{attribute 'monitoring' := 'call'}
PROPERTY Simulated : BOOL
GET
END_GET
END_PROPERTY

{attribute 'monitoring' := 'call'}
PROPERTY Vdc24Okay : BOOL
GET
END_GET
END_PROPERTY

{attribute 'monitoring' := 'call'}
PROPERTY Vdc48Okay : BOOL
GET
END_GET
END_PROPERTY

END_FUNCTION_BLOCK

// _Internal/NullObjects/NullXtsSystemTasks
{attribute 'no_explicit_call' := 'This FB is a CLASS and must be accessed using methods or properties'}
{attribute 'conditionalshow'}
{warning disable C0094}
FUNCTION_BLOCK NullXtsSystemTasks IMPLEMENTS I_XtsTaskCollection, I_NullObject
VAR
END_VAR

METHOD AddTask : BOOL
VAR_INPUT
	Task	: I_XtsTask;
END_VAR
END_METHOD

METHOD CyclicLogic
END_METHOD

METHOD GetTaskById : I_XtsTask
VAR_INPUT
	TaskId	: XtsSystemTaskId;
END_VAR
GetTaskById := NullObjects.XtsTask;
END_METHOD

METHOD GetTaskByName : I_XtsTask
VAR_INPUT
	Name	: T_MaxString;
END_VAR
GetTaskByName := NullObjects.XtsTask;
END_METHOD

METHOD RemoveTaskById
VAR_INPUT
	TaskId	: XtsSystemTaskId;
END_VAR
END_METHOD

METHOD RemoveTaskByInstance
VAR_INPUT
	Task	: I_XtsTask;
END_VAR
END_METHOD

END_FUNCTION_BLOCK

// _Internal/NullObjects/NullXtsTrackCollection
{attribute 'no_explicit_call' := 'This FB is a CLASS and must be accessed using methods or properties'}
{attribute 'conditionalshow'}
{warning disable C0094}
{warning disable C0568}
FUNCTION_BLOCK NullXtsTrackCollection IMPLEMENTS I_XtsTrackCollection, I_NullObject
VAR
END_VAR

METHOD Clear
END_METHOD

PROPERTY Count : UDINT
GET
END_GET
END_PROPERTY

{attribute 'hide'}
METHOD Create : BOOL
VAR_INPUT
	NumberOfTracks : UINT;
END_VAR
END_METHOD

{attribute 'monitoring' := 'call'}
PROPERTY Current : I_XtsTrack
GET
Current := NullObjects.XtsTrack;
END_GET
END_PROPERTY

{attribute 'monitoring' := 'call'}
PROPERTY CurrentIndex : UDINT
GET
END_GET
END_PROPERTY

METHOD GetById : I_XtsTrack
VAR_INPUT
	TrackId : UDINT;
END_VAR
GetById := NullObjects.XtsTrack;
END_METHOD

METHOD GetByOtcid : I_XtsTrack
VAR_INPUT
	TrackOtcid : OTCID;
END_VAR
GetByOtcid := NullObjects.XtsTrack;
END_METHOD

{attribute 'monitoring' := 'call'}
PROPERTY IsEmpty : BOOL
GET
END_GET
END_PROPERTY

PROPERTY MoveToNext : BOOL
GET
END_GET
END_PROPERTY

METHOD ResetIterator
END_METHOD

END_FUNCTION_BLOCK

// _Internal/NullObjects/NullXtsZone
{attribute 'no_explicit_call' := 'This FB is a CLASS and must be accessed using methods or properties'}
{attribute 'conditionalshow'}
{warning disable C0094}
{warning disable C0568}
FUNCTION_BLOCK NullXtsZone IMPLEMENTS I_XtsZone, I_NullObject
VAR
END_VAR

METHOD Accept
VAR_INPUT
	ComponentVisitor	: Core.I_ComponentVisitor;
END_VAR
END_METHOD

METHOD AcceptMoverVisitor
VAR_INPUT
	MoverVisitor : I_XtsMoverVisitor;
END_VAR
END_METHOD

METHOD AcceptXtsZoneVisitor
VAR_INPUT
	ZoneVisitor : I_XtsZoneVisitor;
END_VAR
END_METHOD

{attribute 'monitoring':='call'}
PROPERTY CommandLog : I_XtsLocalLog
GET
CommandLog := NullObjects.MechatronicsLocalLog;
END_GET
END_PROPERTY

METHOD DeregisterWithParent
VAR_INPUT
	Parent	: Core.I_ContainComponents;
END_VAR
END_METHOD

PROPERTY EndPosition : LREAL
GET
END_GET
SET
END_SET
END_PROPERTY

//Select the Nth Mover in the Zone
METHOD GetSortedMover : I_XtsMover
VAR_INPUT
	Index	  : UDINT; // 1 based index
	Direction : Tc3_Mc3Definitions.MC_DIRECTION := Tc3_Mc3Definitions.MC_DIRECTION.mcDirectionPositive; //Direction to fetch from
END_VAR
END_METHOD

METHOD IsMoverInZone : BOOL
VAR_INPUT
	Mover : I_XtsMover;
END_VAR
END_METHOD

PROPERTY Length : LREAL
GET
END_GET
END_PROPERTY

PROPERTY MonitoredMovers : I_XtsMoverCollection
SET
END_SET
END_PROPERTY

PROPERTY Movers : I_XtsMoverEnumerator
GET
Movers := NullObjects.XtsMoverList;
END_GET
END_PROPERTY

PROPERTY Name : Core.T_MaxString
GET
Name := 'Null Xts Zone';
END_GET
SET
END_SET
END_PROPERTY

METHOD RegisterWithParent
VAR_INPUT
	Parent	: Core.I_ContainComponents;
END_VAR
END_METHOD

PROPERTY StartPosition : LREAL
GET
END_GET
SET
END_SET
END_PROPERTY

{attribute 'monitoring':='call'}
PROPERTY Status : I_XtsZoneStatus
GET
Status := NullObjects.XtsZoneStatus;
END_GET
END_PROPERTY

PROPERTY TracePublisher : I_XtsTracePublisher
GET
TracePublisher := NullObjects.MechatronicsTracePublisher;
END_GET
END_PROPERTY

END_FUNCTION_BLOCK

// _Internal/Zone/Status/XtsZoneStatus
{attribute 'no_explicit_call' := 'This FB is a CLASS and must be accessed using methods or properties'}
FUNCTION_BLOCK XtsZoneStatus IMPLEMENTS I_XtsZoneStatus
VAR
	_Zone	: I_XtsZone;
	_Movers : I_XtsMoverCollection;
END_VAR

//FB_Init is always available implicitly and it is used primarily for initialization.

//The return value is not evaluated. For a specific influence, you can also declare the

//methods explicitly and provide additional code there with the standard initialization

//code. You can evaluate the return value.
METHOD FB_Init : BOOL
VAR_INPUT
	bInitRetains : BOOL; // TRUE: the retain variables are initialized (reset warm / reset cold)
	bInCopyCode	 : BOOL; // TRUE: the instance will be copied to the copy code afterward (online change)   
	Zone		 : I_XtsZone;
END_VAR
_Zone := Zone;
END_METHOD

{attribute 'monitoring' := 'call'}
//Number of Movers Currently in Zone
PROPERTY NumberOfMoversInZone : UDINT
GET
NumberOfMoversInZone := _Movers.Count;
END_GET
END_PROPERTY

METHOD SetMoverCollection
VAR_INPUT
	MoverCollection : I_XtsMoverCollection;
END_VAR
_Movers := MoverCollection;
END_METHOD

END_FUNCTION_BLOCK

// _Internal/NullObjects/NullXtsZoneStatus
{attribute 'no_explicit_call' := 'This FB is a CLASS and must be accessed using methods or properties'}
{attribute 'conditionalshow'}
{warning disable C0094}
FUNCTION_BLOCK NullXtsZoneStatus IMPLEMENTS I_XtsZoneStatus, I_NullObject
VAR
END_VAR

{attribute 'monitoring' := 'call'}
PROPERTY NumberOfMoversInZone : UDINT
GET
END_GET
END_PROPERTY

END_FUNCTION_BLOCK

// _Internal/NullObjects/NullZoneCollection
{attribute 'no_explicit_call' := 'This FB is a CLASS and must be accessed using methods or properties'}
{attribute 'conditionalshow'}
{warning disable C0094}
{warning disable C0568}
FUNCTION_BLOCK NullZoneCollection IMPLEMENTS I_XtsZoneCollection, I_NullObject
VAR
END_VAR

METHOD AddItem
VAR_INPUT
	Zone	: I_XtsZone;
END_VAR
END_METHOD

METHOD Clear
END_METHOD

PROPERTY Count : UDINT
GET
END_GET
END_PROPERTY

PROPERTY Current : I_XtsZone
GET
Current := NullObjects.XtsZone;
END_GET
END_PROPERTY

PROPERTY CurrentItem : UDINT
GET
END_GET
END_PROPERTY

{attribute 'monitoring' := 'call'}
PROPERTY IsEmpty : BOOL
GET
END_GET
END_PROPERTY

PROPERTY MoveToNext : BOOL
GET
END_GET
END_PROPERTY

METHOD Remove
VAR_INPUT
	Zone	: I_XtsZone;
END_VAR
END_METHOD

METHOD ResetIterator
END_METHOD

END_FUNCTION_BLOCK

// XtsZone/XtsZone
{attribute 'no_explicit_call' := 'This FB is a CLASS and must be accessed using methods or properties'}
FUNCTION_BLOCK XtsZone EXTENDS CyclicComponent IMPLEMENTS I_XtsZone
VAR
	{attribute 'hide'}
	_Status		: XtsZoneStatus(THIS^);
	_Properties : _DefaultZonePropertyBackers;
	{attribute 'hide'}
	_LocalLogger : XtsLocalLogger;
	{attribute 'hide'}
	_Logger				: XtsTracePublisher;
	_DimensionChecker	: SingleDimensionChecker(_Properties.SingleDimensionBacker);
	_MoverComparer		: MoverZoneDistanceComparer(_Properties.SingleDimensionBacker);
	_DefaultZoneMonitor : ZoneMonitor(_DimensionChecker, _MoverComparer, _Properties.SingleDimensionBacker, _Logger);
	_ZoneMonitor		: I_ZoneMonitor := _DefaultZoneMonitor;
	{attribute 'hide'}
	LogSource : TraceSourceInfo;
	{attribute 'hide'}
	LogMessage : TraceMessageInfo;
END_VAR

//FB_Init is always available implicitly and it is used primarily for initialization.

//The return value is not evaluated. For a specific influence, you can also declare the

//methods explicitly and provide additional code there with the standard initialization

//code. You can evaluate the return value.
METHOD FB_Init : BOOL
VAR_INPUT
	bInitRetains	: BOOL;				 // TRUE: the retain variables are initialized (reset warm / reset cold)
	bInCopyCode		: BOOL;				 // TRUE: the instance will be copied to the copy code afterward (online change)   
	Name			: T_MaxString;		 //Name of the Zone
	MonitoredMovers : I_XtsMoverCollection; //Collection of Movers for the Zone to monitor
	StartPosition	: LREAL := 0;		 //Start position of the Zone in mm
	EndPosition		: LREAL := 0;		 //End position of the Zone in mm
	System			: I_ContainXtsZones; //XtsSystem to self register to
END_VAR
_ZoneMonitor.MonitoredMovers := MonitoredMovers;
LogSource.SourceName		 := 'Zone Object';
_Logger.Subscribe(_LocalLogger);
IF XtsCoreParameters.TcEventLoggerEnabled THEN
	_Logger.Subscribe(XtsTrace.EventLogger);
END_IF

_Status.SetMoverCollection(_ZoneMonitor.Movers);
THIS^.StartPosition := StartPosition;
THIS^.EndPosition	:= EndPosition;
IF System <> 0 THEN
	System.Zones.AddItem(THIS^);
	RegisterWithParent(System);
END_IF
END_METHOD

{attribute 'monitoring':='call'}
//End Position of the Zone in mm
PROPERTY EndPosition : LREAL
GET
EndPosition := _Properties.SingleDimensionBacker.EndPosition;
END_GET
SET
_Properties.SingleDimensionBacker.EndPosition := EndPosition;
END_SET
END_PROPERTY

{attribute 'monitoring':='call'}
//Start Position of the Zone in mm
PROPERTY StartPosition : LREAL
GET
StartPosition := _Properties.SingleDimensionBacker.StartPosition;
END_GET
SET
_Properties.SingleDimensionBacker.StartPosition := StartPosition;
END_SET
END_PROPERTY

{attribute 'monitoring':='call'}
PROPERTY CommandLog : I_XtsLocalLog
GET
CommandLog := _LocalLogger;
END_GET
END_PROPERTY

PROPERTY TracePublisher : I_XtsTracePublisher
GET
TracePublisher := _Logger;
END_GET
END_PROPERTY

METHOD AcceptMoverVisitor
VAR_INPUT
	MoverVisitor	: I_XtsMoverVisitor;
END_VAR
_ZoneMonitor.Movers.AcceptMoverVisitor(MoverVisitor);
END_METHOD

METHOD AcceptXtsZoneVisitor
VAR_INPUT
	ZoneVisitor : I_XtsZoneVisitor;
END_VAR
ZoneVisitor.VisitZone(THIS^);
END_METHOD

METHOD CyclicLogic
VAR
	Mover : I_XtsMover;
END_VAR
_ZoneMonitor.CyclicLogic();
END_METHOD

//Select the Nth Mover in the Zone
METHOD GetSortedMover : I_XtsMover
VAR_INPUT
	Index	  : UDINT; // 1 based index
	Direction : Tc3_Mc3Definitions.MC_DIRECTION := Tc3_Mc3Definitions.MC_DIRECTION.mcDirectionPositive; //Direction to fetch from
END_VAR
VAR
	DesiredIndex : UDINT;
END_VAR
GetSortedMover := NullObjects.XtsMover;
IF Index <= 0 OR Index > _ZoneMonitor.Movers.Count THEN
	LogMessage.Message	 := 'GetSortedMover Requested Index Out of bounds';
	LogMessage.Severity	 := 2;
	LogMessage.MessageId := E_XtsLogMessage.ZoneMoverErrorGetSortedIndexOOB;
	_Logger.LogMessageInstance(LogSource, LogMessage);
	RETURN;
END_IF

IF Direction = Tc3_Mc3Definitions.MC_Direction.mcDirectionNegative THEN
	DesiredIndex := _ZoneMonitor.Movers.Count - Index;
ELSE
	DesiredIndex := Index - 1;
END_IF

GetSortedMover := _ZoneMonitor.Movers.GetAtIndex(DesiredIndex);
END_METHOD

//Check if Mover is currently in Zone
METHOD IsMoverInZone : BOOL
VAR_INPUT
	Mover : I_XtsMover; //Mover to check
END_VAR
IsMoverInZone := _ZoneMonitor.Movers.Contains(Mover);
END_METHOD

//Movers currently monitored by Zone
PROPERTY MonitoredMovers : I_XtsMoverCollection
SET
_ZoneMonitor.MonitoredMovers := MonitoredMovers;
END_SET
END_PROPERTY

//Movers currently in the Zone
PROPERTY Movers : I_XtsMoverEnumerator
GET
Movers := _ZoneMonitor.Movers;
END_GET
END_PROPERTY

{attribute 'monitoring':='call'}
PROPERTY Status : I_XtsZoneStatus
GET
Status := _Status;
END_GET
END_PROPERTY

END_FUNCTION_BLOCK

// _Internal/Zone/Properties/_DefaultZonePropertyBackers
{attribute 'no_explicit_call' := 'This FB is a CLASS and must be accessed using methods or properties'}
FUNCTION_BLOCK _DefaultZonePropertyBackers
VAR
	_DefaultSingleDimensionZone : SingleDimensionZone;
	//
	_SingleDimensionZone : I_SingleDimensionZone := _DefaultSingleDimensionZone;
END_VAR

{attribute 'monitoring':='call'}
PROPERTY SingleDimensionBacker : I_SingleDimensionZone
GET
SingleDimensionBacker := _SingleDimensionZone;
END_GET
SET
_SingleDimensionZone := SingleDimensionBacker;
END_SET
END_PROPERTY

END_FUNCTION_BLOCK

// _Internal/Zone/Properties/SingleDimensionZone
{attribute 'no_explicit_call' := 'This FB is a CLASS and must be accessed using methods or properties'}
FUNCTION_BLOCK SingleDimensionZone IMPLEMENTS I_SingleDimensionZone
VAR
	_StartPosition : LREAL;
	_EndPosition   : LREAL;
END_VAR

{attribute 'monitoring':='call'}
PROPERTY EndPosition : LREAL
GET
EndPosition := _EndPosition;
END_GET
SET
_EndPosition := EndPosition;
END_SET
END_PROPERTY

{attribute 'monitoring':='call'}
PROPERTY StartPosition : LREAL
GET
StartPosition := _StartPosition;
END_GET
SET
_StartPosition := StartPosition;
END_SET
END_PROPERTY

END_FUNCTION_BLOCK

// _Internal/Zone/SingleDimensionChecker
{attribute 'no_explicit_call' := 'This FB is a CLASS and must be accessed using methods or properties'}
{attribute 'conditional_show'}
FUNCTION_BLOCK SingleDimensionChecker IMPLEMENTS I_MoverInPositionChecker
VAR
	_Dimensions : I_SingleDimensionZone;
END_VAR

//FB_Init is always available implicitly and it is used primarily for initialization.

//The return value is not evaluated. For a specific influence, you can also declare the

//methods explicitly and provide additional code there with the standard initialization

//code. You can evaluate the return value.
METHOD FB_Init : BOOL
VAR_INPUT
	bInitRetains : BOOL; // TRUE: the retain variables are initialized (reset warm / reset cold)
	bInCopyCode	 : BOOL; // TRUE: the instance will be copied to the copy code afterward (online change)  
	Dimensions	 : I_SingleDimensionZone;
END_VAR
_Dimensions := Dimensions;
END_METHOD

METHOD IsMoverInPosition : BOOL
VAR_INPUT
	Mover : I_XtsMover;
END_VAR

VAR
	startPosition : LREAL;
	endPosition	  : LREAL;
	tmp : LREAL;
END_VAR
startPosition := _Dimensions.StartPosition;
endPosition	  := _Dimensions.EndPosition;
IF Mover.Status.CurrentTrack.Length <> 0 THEN
	startPosition := startPosition - Mover.Status.CurrentTrack.Length * TRUNC(_Dimensions.StartPosition / Mover.Status.CurrentTrack.Length);
	IF startPosition < 0.0 THEN
		startPosition := startPosition + Mover.Status.CurrentTrack.Length;
	END_IF

	endPosition := endPosition - Mover.Status.CurrentTrack.Length * TRUNC(_Dimensions.EndPosition / Mover.Status.CurrentTrack.Length);
	IF endPosition < 0.0 THEN
		endPosition := endPosition + Mover.Status.CurrentTrack.Length;
	END_IF
END_IF

IF startPosition < endPosition THEN
	IsMoverInPosition := Mover.Position > startPosition AND Mover.Position < endPosition;
ELSE
	IsMoverInPosition := Mover.Position > startPosition OR Mover.Position < endPosition;
END_IF
END_METHOD

END_FUNCTION_BLOCK

// _Internal/Zone/Interfaces/I_MoverInPositionChecker
INTERFACE I_MoverInPositionChecker EXTENDS I_Base

METHOD IsMoverInPosition : BOOL
VAR_INPUT
	Mover : I_XtsMover;
END_VAR
END_METHOD

END_INTERFACE

// _Internal/Zone/MoverZoneDistanceComparer
{attribute 'no_explicit_call' := 'This FB is a CLASS and must be accessed using methods or properties'}
{attribute 'conditional_show'}
FUNCTION_BLOCK MoverZoneDistanceComparer IMPLEMENTS I_XtsMoverComparer
VAR
	_ZoneDimensions : I_SingleDimensionZone;
END_VAR

METHOD Compare : SINT
VAR_INPUT
	Mover1 : I_XtsMover;
	Mover2 : I_XtsMover;
END_VAR

VAR
	Mover1Distance : LREAL;
	Mover2Distance : LREAL;
END_VAR
Mover1Distance := MoverDistance(_ZoneDimensions.StartPosition, Mover1.Position, Mover1.Status.CurrentTrack.Length);
Mover2Distance := MoverDistance(_ZoneDimensions.StartPosition, Mover2.Position, Mover2.Status.CurrentTrack.Length);
IF Mover1Distance < Mover2Distance THEN
	Compare := -1;
ELSIF Mover1Distance > Mover2Distance THEN
	Compare := 1;
ELSE
	Compare := 0;
END_IF
END_METHOD

//FB_Init is always available implicitly and it is used primarily for initialization.
//The return value is not evaluated. For a specific influence, you can also declare the
//methods explicitly and provide additional code there with the standard initialization
//code. You can evaluate the return value.
METHOD FB_Init: BOOL
VAR_INPUT
    bInitRetains: BOOL; // TRUE: the retain variables are initialized (reset warm / reset cold)
    bInCopyCode: BOOL;  // TRUE: the instance will be copied to the copy code afterward (online change)   
	Dimensions : I_SingleDimensionZone;
END_VAR
_ZoneDimensions := Dimensions;
END_METHOD

END_FUNCTION_BLOCK

// _Internal/Zone/Interfaces/I_XtsMoverComparer
INTERFACE I_XtsMoverComparer EXTENDS I_Base

METHOD Compare : SINT
VAR_INPUT
	Mover1 : I_XtsMover;
	Mover2 : I_XtsMover;
END_VAR
END_METHOD

END_INTERFACE

// _Internal/Zone/MoverDistance
FUNCTION MoverDistance : LREAL
VAR_INPUT
	StartPosition : LREAL;
	MoverPosition : LREAL;
	TrackLength	  : LREAL;
END_VAR

VAR
	NormalizedStart : LREAL;
	Distance		: LREAL;
END_VAR

IF TrackLength = 0 THEN
	MoverDistance := 0;
	RETURN;
END_IF

NormalizedStart := StartPosition - TrackLength * TRUNC(StartPosition / TrackLength);
IF normalizedStart < 0 THEN
	NormalizedStart := NormalizedStart + TrackLength;
END_IF;

Distance := MoverPosition - NormalizedStart;
IF Distance < 0 THEN
	Distance := Distance + TrackLength;
END_IF;

MoverDistance := Distance;

END_FUNCTION

// _Internal/Zone/ZoneMonitor
{attribute 'no_explicit_call' := 'This FB is a CLASS and must be accessed using methods or properties'}
{attribute 'conditional_show'}
FUNCTION_BLOCK ZoneMonitor IMPLEMENTS I_ZoneMonitor
VAR
	_DefaultCurrentMovers : XtsMoverList;
	_CurrentMovers		  : I_XtsMoverList := _DefaultCurrentMovers;
	_MoverChecker		  : I_MoverInPositionChecker;
	_MonitoredMovers	  : I_XtsMoverCollection;
	_ZoneComparer		  : I_XtsMoverComparer;
	_ZoneDimensions		  : I_SingleDimensionZone;
	_Logger				  : I_XtsLogger;
	LogSource			  : TraceSourceInfo;
	LogMessage			  : TraceMessageInfo;
END_VAR

METHOD CyclicLogic
VAR
	Mover				   : I_XtsMover;
	inPosition			   : BOOL;
	inCollection		   : BOOL;
	additionIndex		   : UDINT;
	CompareResults		   : SINT;
	EntranceEvent		   : E_ThresholdEvent;
	ExitEvent			   : E_ThresholdEvent;
	ThresholdEventOccurred : BOOL;
END_VAR
_MonitoredMovers.ResetIterator();
WHILE _MonitoredMovers.MoveToNext DO
	__QUERYINTERFACE(_MonitoredMovers.Current, Mover);
	IF Mover.Status.CurrentTrack.Length = 0 THEN
		LogMessage.MessageId := E_XtsLogMessage.ZoneMoverErrorTrackLengthZero;
		LogMessage.Message	 := CONCAT(Mover.Name, ' current Track Length 0 unable to add to track');
		LogMessage.Severity	 := 3;
		_Logger.LogMessageInstance(LogSource, LogMessage);
		CONTINUE;
	END_IF

	inPosition := _MoverChecker.IsMoverInPosition(Mover);

	//Need to check if crossed the threshold of the exit or the entrance
	EntranceEvent		   := CheckForThresholdEvent(Mover, _ZoneDimensions.StartPosition);
	ExitEvent			   := CheckForThresholdEvent(Mover, _ZoneDimensions.EndPosition);
	ThresholdEventOccurred := (EntranceEvent <> E_ThresholdEvent.NoEvent) AND (ExitEvent <> E_ThresholdEvent.NoEvent);
	inCollection		   := _CurrentMovers.Contains(Mover);
	IF NOT inPosition AND inCollection THEN
		_CurrentMovers.Remove(Mover);
		CONTINUE;
	END_IF

	//Adds the Mover into the collection sorted by Position Descending
	IF inPosition AND NOT inCollection THEN
		_CurrentMovers.ResetIterator();
		WHILE _CurrentMovers.MoveToNext DO
			CompareResults := _ZoneComparer.Compare(Mover, _CurrentMovers.Current);
			IF CompareResults < 0 THEN //Mover 1 is closer to Start
				additionIndex := _CurrentMovers.CurrentItem - 1;
				EXIT;
			ELSIF CompareResults > 0 THEN //Mover 2 is closer to Start
				additionIndex := _CurrentMovers.CurrentItem;
			ELSE //Movers are equadistant, should never happen. Only realistically happens if TrackLength = 0

				//
			END_IF
		END_WHILE

		_CurrentMovers.InsertAtIndex(Mover, additionIndex);
	ELSIF ThresholdEventOccurred AND inCollection THEN
		(*Search the Collection to find the new index
			Remove from old index
			Add to new*)
		_CurrentMovers.ResetIterator();
		WHILE _CurrentMovers.MoveToNext DO
			CompareResults := _ZoneComparer.Compare(Mover, _CurrentMovers.Current);
			IF CompareResults < 0 THEN //Mover 1 is closer to Start
				additionIndex := _CurrentMovers.CurrentItem - 1;
				EXIT;
			ELSIF CompareResults > 0 THEN //Mover 2 is closer to Start
				additionIndex := _CurrentMovers.CurrentItem;
			ELSE //Movers are equadistant, should never happen. Only realistically happens if TrackLength = 0

				//
			END_IF
		END_WHILE

		_CurrentMovers.Remove(Mover);
		_CurrentMovers.InsertAtIndex(Mover, additionIndex);
	END_IF
END_WHILE
END_METHOD

//FB_Init is always available implicitly and it is used primarily for initialization.

//The return value is not evaluated. For a specific influence, you can also declare the

//methods explicitly and provide additional code there with the standard initialization

//code. You can evaluate the return value.
METHOD FB_Init : BOOL
VAR_INPUT
	bInitRetains	: BOOL; // TRUE: the retain variables are initialized (reset warm / reset cold)
	bInCopyCode		: BOOL; // TRUE: the instance will be copied to the copy code afterward (online change)   
	PositionChecker : I_MoverInPositionChecker;
	ZoneComparer	: I_XtsMoverComparer;
	ZoneDimensions	: I_SingleDimensionZone;
	Logger			: I_XtsLogger;
END_VAR
_MoverChecker		 := PositionChecker;
_ZoneComparer		 := ZoneComparer;
_Logger				 := Logger;
_ZoneDimensions		 := ZoneDimensions;
LogSource.SourceName := 'ZoneMonitor';
END_METHOD

PROPERTY MonitoredMovers : I_XtsMoverCollection
SET
_MonitoredMovers := MonitoredMovers;
END_SET
END_PROPERTY

{attribute 'monitoring':='call'}
PROPERTY Movers : I_XtsMoverList
GET
Movers := _CurrentMovers;
END_GET
END_PROPERTY

END_FUNCTION_BLOCK

// _Internal/Zone/Interfaces/I_ZoneMonitor
INTERFACE I_ZoneMonitor EXTENDS I_Base, I_Cyclic, I_MonitorsMovers, I_ContainXtsMoverList

END_INTERFACE

// _Internal/Peeker/Interfaces/I_XtsModuleCollectionPeeker
INTERFACE I_XtsModuleCollectionPeeker EXTENDS I_Base

METHOD SetCollection
VAR_INPUT
	NewCollection  : I_XtsModuleCollection;
	CollectionName : T_MaxString := 'A Collection';
END_VAR
END_METHOD

END_INTERFACE

// _Internal/Peeker/Interfaces/I_XtsMoverCollectionPeeker
INTERFACE I_XtsMoverCollectionPeeker EXTENDS I_Base

METHOD SetCollection
VAR_INPUT
	NewCollection  : I_XtsMoverCollection;
	CollectionName : T_MaxString := 'A Collection';
END_VAR
END_METHOD

END_INTERFACE

// _Internal/Peeker/Interfaces/I_XtsPartCollectionPeeker
INTERFACE I_XtsPartCollectionPeeker EXTENDS I_Base

METHOD SetCollection
VAR_INPUT
	NewCollection  : I_XtsPartCollection;
	CollectionName : T_MaxString := 'A Collection';
END_VAR
END_METHOD

END_INTERFACE

// _Internal/Peeker/Interfaces/I_XtsPositionTriggerCollectionPeeker
INTERFACE I_XtsPositionTriggerCollectionPeeker EXTENDS I_Base

METHOD SetCollection
VAR_INPUT
	NewCollection  : I_XtsPositionTriggerCollection;
	CollectionName : T_MaxString := 'A Collection';
END_VAR
END_METHOD

END_INTERFACE

// _Internal/Peeker/Interfaces/I_XtsStationCollectionPeeker
INTERFACE I_XtsStationCollectionPeeker EXTENDS I_Base

METHOD SetCollection
VAR_INPUT
	NewCollection  : I_XtsStationCollection;
	CollectionName : T_MaxString := 'A Collection';
END_VAR
END_METHOD

END_INTERFACE

// _Internal/Peeker/Interfaces/I_XtsZoneCollectionPeeker
INTERFACE I_XtsZoneCollectionPeeker EXTENDS I_Base

METHOD SetCollection
VAR_INPUT
	NewCollection  : I_XtsZoneCollection;
	CollectionName : T_MaxString := 'A Collection';
END_VAR
END_METHOD

END_INTERFACE

// _Internal/Station/Interfaces/I_StationTaskCollection
INTERFACE I_StationTaskCollection EXTENDS I_Base

END_INTERFACE

// _Internal/Station/MoverMonitorTask
{attribute 'no_explicit_call' := 'This FB is a CLASS and must be accessed using methods or properties'}
FUNCTION_BLOCK MoverMonitorTask IMPLEMENTS I_MoverMonitor
VAR
	_MonitoredMovers  : I_XtsMoverCollection;
	_CurrentMover	  : I_XtsMover := NullObjects.XtsMover;
	_RemoveCollection : XtsMoverCollection;
	_Station		  : I_XtsStation;
	{attribute 'hide'}
	_Logger : I_XtsLogger;
	{attribute 'hide'}
	LogSource : TraceSourceInfo;
	{attribute 'hide'}
	LogMessage : TraceMessageInfo;
END_VAR

METHOD CyclicLogic
VAR
	Mover	  : I_XtsMover;
	NullMover : I_XtsMover;
END_VAR
_MonitoredMovers.ResetIterator();
WHILE _MonitoredMovers.MoveToNext DO
	Mover := _MonitoredMovers.Current;
	IF Mover.CurrentTask.TaskId <> MoverTaskID.MOVE_TO_STATION OR Mover.Status.CommandedStation <> _Station THEN
		_RemoveCollection.AddItem(Mover);
		CONTINUE;
	END_IF

	NullMover := NullObjects.XtsMover;
	IF Mover.InPosition AND _CurrentMover = NullMover THEN
		_CurrentMover		 := Mover;
		LogMessage.Message	 := CONCAT(Mover.Name, ' arrived at station');
		LogMessage.MessageId := E_XtsLogMessage.StationMoverArrived;
		LogMessage.Severity	 := 0;
		_Logger.LogMessageInstance(LogSource, LogMessage);
		EXIT;
	END_IF
END_WHILE

IF _RemoveCollection.IsEmpty THEN
	RETURN;
END_IF

_RemoveCollection.ResetIterator();
WHILE _RemoveCollection.MoveToNext DO
	LogMessage.Message	 := CONCAT(_RemoveCollection.Current.Name, ' deregistered from Station');
	LogMessage.MessageId := E_XtsLogMessage.StationMoverDeregistered;
	LogMessage.Severity	 := 0;
	_Logger.LogMessageInstance(LogSource, LogMessage);
	IF _CurrentMover = _RemoveCollection.Current THEN
		_CurrentMover := NullObjects.XtsMover;
	END_IF

	_MonitoredMovers.Remove(_RemoveCollection.Current);
END_WHILE

IF NOT _RemoveCollection.IsEmpty THEN
	_RemoveCollection.Clear();
END_IF
END_METHOD

//FB_Init is always available implicitly and it is used primarily for initialization.

//The return value is not evaluated. For a specific influence, you can also declare the

//methods explicitly and provide additional code there with the standard initialization

//code. You can evaluate the return value.
METHOD FB_Init : BOOL
VAR_INPUT
	bInitRetains			 : BOOL; // TRUE: the retain variables are initialized (reset warm / reset cold)
	bInCopyCode				 : BOOL; // TRUE: the instance will be copied to the copy code afterward (online change)
	Station					 : I_XtsStation;
	MonitoredMoverCollection : I_XtsMoverCollection;
END_VAR
_Station		 := Station;
__QUERYINTERFACE(Station.TracePublisher,_Logger);
LogSource.SourceName := 'Mover Monitor';
_MonitoredMovers := MonitoredMoverCollection;
END_METHOD

METHOD GetMover : I_XtsMover
VAR
	NullMover : I_XtsMover;
END_VAR
NullMover := NullObjects.XtsMover;
IF _CurrentMover = NullMover THEN
	LogMessage.Message	 := 'GetMover called when no mover present.';
	LogMessage.Severity	 := 2;
	LogMessage.MessageId := E_XtsLogMessage.StationGetMoverCalledNoMover;
	_Logger.LogMessageInstance(LogSource, LogMessage);
	GetMover := NullObjects.XtsMover;
	RETURN;
END_IF

GetMover := _CurrentMover;
_MonitoredMovers.Remove(_CurrentMover);
_CurrentMover := NullObjects.XtsMover;
END_METHOD

PROPERTY MonitoredMovers : I_XtsMoverCollection
GET
MonitoredMovers := _MonitoredMovers;
END_GET
SET
_MonitoredMovers := MonitoredMovers;
END_SET
END_PROPERTY

{attribute 'monitoring':='call'}
PROPERTY MoverPresent : BOOL
GET
VAR
	NullMover : I_XtsMover;
END_VAR
NullMover	 := NullObjects.XtsMover;
MoverPresent := _CurrentMover <> NullMover;
END_GET
END_PROPERTY

END_FUNCTION_BLOCK

// _Internal/Tracing/XtsCoreEventLogger
{attribute 'no_explicit_call' := 'This FB is a CLASS and must be accessed using methods or properties'}
{attribute 'conditional_show'}
FUNCTION_BLOCK XtsCoreEventLogger IMPLEMENTS I_XtsLogger
VAR
	MessagesThisScan : DINT;
	Message			 : FB_TcMessage;
	Source			 : FB_TcSourceInfo;
	CurrentCycle	 : UDINT;
END_VAR

METHOD LogMessage
VAR_INPUT
	Key		  : T_MaxString;
	Value	  : T_MaxString;
	SourceId  : UDINT := 0;
	TimeStamp : ULINT := 0;
	MessageId : UDINT := 1;
	Severity  : USINT := 1;
END_VAR

VAR_INST
	LogSource  : TraceSourceInfo;
	LogMessage : TraceMessageInfo;
END_VAR
LogSource.SourceName := Key;
LogSource.SourceId	 := SourceId;
LogSource.TimeStamp	 := TimeStamp;
LogMessage.Message	 := Value;
LogMessage.MessageId := MessageId;
LogMessage.Severity	 := Severity;
THIS^.LogMessageInstance(LogSource, LogMessage);
END_METHOD

METHOD LogMessageInstance
VAR_INPUT
	SourceInfo	: I_TraceSourceInfo;
	MessageInfo : I_TraceMessageInfo;
	Arguments	: I_TraceArgument := 0;
END_VAR
VAR
	Msg : T_MaxString;
END_VAR
IF TwinCAT_SystemInfoVarList._TaskInfo[GETCURTASKINDEXEX()].CycleCount <> CurrentCycle THEN
	CurrentCycle	 := TwinCAT_SystemInfoVarList._TaskInfo[GETCURTASKINDEXEX()].CycleCount;
	MessagesThisScan := 0;
END_IF

IF MessagesThisScan < TO_DINT(TwinCAT_SystemInfoVarList._TaskInfo[GETCURTASKINDEXEX()].CycleTime / 2000) THEN
	Source.sName := SourceInfo.SourceName;
	Source.nId	 := SourceInfo.SourceId;
	Message.Create(eventClass	:= TC_EVENT_CLASSES.XtsCoreEvents,
				   nEventId		:= MessageInfo.MessageId,
				   eSeverity	:= USINT_To_TcEventSeverity(MessageInfo.Severity),
				   ipSourceInfo := Source);

	Msg := MessageInfo.Message;
	Message.ipArguments.Clear().AddString(Msg);
	Message.Send(0);
	Message.Release();
	Source.Clear();
	MessagesThisScan := MessagesThisScan + 1;
END_IF
END_METHOD

END_FUNCTION_BLOCK

// _Internal/Zone/Properties/_DefaultZoneProperties
{attribute 'no_explicit_call' := 'This FB is a CLASS and must be accessed using methods or properties'}
FUNCTION_BLOCK _DefaultZoneProperties
VAR
	_DefaultSingleDimensionZone : SingleDimensionZone;
END_VAR

END_FUNCTION_BLOCK

// HMI/XtsBasicHmi
{attribute 'no_explicit_call' := 'This FB is a CLASS and must be accessed using methods or properties'}
FUNCTION_BLOCK XtsBasicHmi
VAR_GENERIC CONSTANT
	MaxNumberOfMovers			: UDINT := 1;
	MaxNumberOfStations			: UDINT := 1;
	MaxNumberOfPositionTriggers : UDINT := 1;
	MaxNumberOfZones			: UDINT := 1;
END_VAR
EXTENDS HmiFunction IMPLEMENTS I_ModuleVisitor, I_ComponentVisitor
VAR CONSTANT
	TotalCyclicRunner : UDINT := MaxNumberOfMovers + MaxNumberOfStations + MaxNumberOfPositionTriggers + MaxNumberOfZones + 1;
END_VAR

VAR
	_System					   : I_XtsSystem;
	_Built					   : BOOL;
	_CyclicRunner			   : CyclicRunner<TotalCyclicRunner>;
	_MoverCount				   : UINT;
	_StationCount			   : UINT;
	_PositionTriggerCount	   : UINT;
	_ZoneCount				   : UINT;
	_MoverHmiObjects		   : ARRAY[1..MaxNumberOfMovers] OF XtsMover_HMI('Name', 0);
	_StationHmiObjects		   : ARRAY[1..MaxNumberOfStations] OF XtsStation_HMI('Name', 0);
	_PositionTriggerHmiObjects : ARRAY[1..MaxNumberOfPositionTriggers] OF XTSPositionTrigger_HMI('Name', 0);
	_ZoneHmiObjects			   : ARRAY[1..MaxNumberOfZones] OF XtsZone_HMI('Name', 0);
	_SystemHmi				   : XtsSystem_HMI('Name', 0);
END_VAR

(*FB_Init is always available implicitly and it is used primarily for initialization.
The return value is not evaluated. For a specific influence, you can also declare the
methods explicitly and provide additional code there with the standard initialization
code. You can evaluate the return value.*)
METHOD FB_Init : BOOL
VAR_INPUT
	(* TRUE: the retain variables are initialized (reset warm / reset cold)*)
	bInitRetains : BOOL;

	(* TRUE: the instance will be copied to the copy code afterward (online change)   *)
	bInCopyCode : BOOL;
	Name		: Core.T_MaxString;
	System		: I_XtsSystem;
END_VAR
VAR
	i : UDINT;
END_VAR
ControlType				 := 'XtsSystem';
LinkObject				 := 'Xts_HMI';
_System					 := System;
_SystemHmi.ControlObject := _System;
_SystemHmi.Name			 := _System.Name;
_CyclicRunner.AddCallee(_SystemHmi);
FOR i := 1 TO MaxNumberOfMovers DO
	_CyclicRunner.AddCallee(_MoverHmiObjects[i]);
END_FOR

FOR i := 1 TO MaxNumberOfStations DO
	_CyclicRunner.AddCallee(_StationHmiObjects[i]);
END_FOR

FOR i := 1 TO MaxNumberOfPositionTriggers DO
	_CyclicRunner.AddCallee(_PositionTriggerHmiObjects[i]);
END_FOR

FOR i := 1 TO MaxNumberOfZones DO
	_CyclicRunner.AddCallee(_ZoneHmiObjects[i]);
END_FOR
END_METHOD

METHOD Accept
VAR_INPUT
	ComponentVisitor	: Core.I_ComponentVisitor;
END_VAR
VAR
	i : UDINT;
END_VAR
FOR i := 1 TO MaxNumberOfMovers DO
	_MoverHmiObjects[i].Accept(ComponentVisitor);
END_FOR

FOR i := 1 TO MaxNumberOfStations DO
	_StationHmiObjects[i].Accept(ComponentVisitor);
END_FOR

FOR i := 1 TO MaxNumberOfPositionTriggers DO
	_PositionTriggerHmiObjects[i].Accept(ComponentVisitor);
END_FOR

FOR i := 1 TO MaxNumberOfZones DO
	_ZoneHmiObjects[i].Accept(ComponentVisitor);
END_FOR
END_METHOD

METHOD BuildHMI : BOOL
VAR_INPUT
END_VAR
IF _Built THEN
	RETURN;
END_IF

_System.Accept(THIS^);
_Built	 := TRUE;
BuildHMI := TRUE;
END_METHOD

PROPERTY ControlObject : I_Base
SET
_SystemHmi.ControlObject := ControlObject;
__QUERYINTERFACE(ControlObject, _System);
_SystemHmi.Name := _System.Name;
END_SET
END_PROPERTY

METHOD CyclicLogic
IF _System = 0 THEN
	RETURN;
END_IF

_CyclicRunner.CallAll();
END_METHOD

METHOD VisitComponent
VAR_INPUT
	Component : I_Component;
END_VAR

VAR
	_XtsStation			: I_XtsStation;
	_XtsPositionTrigger : I_XtsPositionTrigger;
	_XtsMover			: I_XtsMover;
	_XtsZone			: I_XtsZone;
END_VAR
IF __QUERYINTERFACE(Component, _XtsMover) THEN
	_MoverCount									:= _MoverCount + 1;
	_MoverHmiObjects[_MoverCount].ControlObject := _XtsMover;
	_MoverHmiObjects[_MoverCount].Name			:= _XtsMover.Name;
ELSIF __QUERYINTERFACE(Component, _XtsPositionTrigger) THEN
	_PositionTriggerCount											:= _PositionTriggerCount + 1;
	_PositionTriggerHmiObjects[_PositionTriggerCount].ControlObject := _XtsPositionTrigger;
	_PositionTriggerHmiObjects[_PositionTriggerCount].Name			:= _XtsPositionTrigger.Name;
ELSIF __QUERYINTERFACE(Component, _XtsStation) THEN
	_StationCount									:= _StationCount + 1;
	_StationHmiObjects[_StationCount].ControlObject := _XtsStation;
	_StationHmiObjects[_StationCount].Name			:= _XtsStation.Name;
ELSIF __QUERYINTERFACE(Component, _XtsZone) THEN
	_ZoneCount								  := _ZoneCount + 1;
	_ZoneHmiObjects[_ZoneCount].ControlObject := _XtsZone;
	_ZoneHmiObjects[_ZoneCount].Name		  := _XtsZone.Name;
END_IF
END_METHOD

METHOD VisitModule
VAR_INPUT
	Module : I_Module;
END_VAR

VAR
	_XtsPart	: I_XtsPart;
END_VAR
Module.Components.Accept(THIS^);
Module.Modules.Accept(THIS^);
END_METHOD

END_FUNCTION_BLOCK

// HMI/XtsMover_HMI
FUNCTION_BLOCK XtsMover_HMI EXTENDS HmiFunction
VAR
	Mover : I_XtsMover;
	{ attribute 'TcHmiSymbol.AddSymbol' }
	{ attribute 'TcHmiSymbol.AddSymbol.UserGroups' := '__SystemAdministrators,Admin' }
	Mover_HMI : ST_XtsMover_HMI;
END_VAR

PROPERTY ControlObject : I_Base
SET
__QUERYINTERFACE(ControlObject, Mover);
END_SET
END_PROPERTY

METHOD CyclicLogic
VAR_INST
	EnableRT	  : R_TRIG;
	DisableRT	  : R_TRIG;
	ResetRT		  : R_TRIG;
	ClearLogRT	  : R_TRIG;
	MovePosRT	  : R_TRIG;
	MoveVeloRT	  : R_Trig;
	MoveStationRT : R_TRIG;
	BumpCommandRT : R_TRIG;
	HaltRT		  : R_TRIG;
END_VAR
IF Mover = 0 THEN
	RETURN;
END_IF

Mover_Hmi.Enabled			:= Mover.Enabled;
Mover_Hmi.Busy				:= Mover.Busy;
Mover_HMI.Acceleration		:= Mover.Status.SetAcceleration;
Mover_HMI.Velocity			:= Mover.Status.SetVelocity;
Mover_HMI.Deceleration		:= Mover.Parameters.Deceleration;
Mover_HMI.Jerk				:= Mover.Parameters.Jerk;
Mover_HMI.Gap				:= Mover.Parameters.Gap;
Mover_HMI.Initialized		:= Mover.Initialized;
Mover_HMI.HasError			:= Mover.Error;
Mover_HMI.ErrorId			:= Mover.ErrorId;
Mover_HMI.Position			:= Mover.Position;
Mover_HMI.Id				:= Mover.MoverId;
Mover_HMI.Name				:= Mover.Name;
Mover_HMI.IdentInGroup		:= Mover.Status.IdentInGroup;
Mover_HMI.LocalLog.Logs		:= Mover.CommandLog.Commands;
Mover_HMI.AvoidingCollision := Mover.Status.AvoidingCollision;
IF Mover.Busy THEN
	Mover_HMI.CurrentTask := Mover.CurrentTask.TaskName;
ELSE
	Mover_HMI.CurrentTask := '';
END_IF

Mover_HMI.CommandedPosition	   := Mover.Status.CommandedPosition;
Mover_HMI.CommandedStationName := Mover.Status.CommandedStation.Name;
//Commands from HMI disabled if the HMI is not enabled
IF NOT Mover_HMI.HmiEnabled THEN
	RETURN;
END_IF

ClearLogRT(Clk := Mover_HMI.LocalLog.ClearLog);
IF ClearLogRT.Q THEN
	Mover.CommandLog.Clear();
END_IF

Mover_HMI.Commands.Enable.Permissive.Set(0, 'Mover enabled', NOT Mover.Enabled);
EnableRT(Clk := Mover_HMI.Commands.Enable.Active);
IF EnableRT.Q AND NOT Mover.Enabled THEN
	Mover.Enable();
END_IF

Mover_HMI.Commands.Disable.Permissive.Set(0, 'Mover not enabled', Mover.Enabled);
DisableRT(Clk := Mover_HMI.Commands.Disable.Active);
IF DisableRT.Q THEN
	Mover.Disable();
END_IF

Mover_HMI.Commands.MoveVelocity.Permissive.Set(0, 'Mover not enabled', Mover.Enabled);
MoveVeloRT(Clk := Mover_HMI.Commands.MoveVelocity.Active);
IF MoveVeloRT.Q THEN
	Mover.Parameters.Acceleration := Mover_HMI.Parameters.Acceleration;
	Mover.Parameters.Deceleration := Mover_HMI.Parameters.Deceleration;
	Mover.Parameters.Jerk		  := Mover_HMI.Parameters.Jerk;
	Mover.Parameters.Gap		  := Mover_HMI.Parameters.Gap;
	Mover.MoveVelocity(Velocity := Mover_HMI.Parameters.Velocity);
END_IF

Mover_HMI.Commands.MoveToPosition.Permissive.Set(0, 'Mover not enabled', Mover.Enabled);
MovePosRt(Clk := Mover_Hmi.Commands.MoveToPosition.Active);
IF MovePosRt.Q THEN
	Mover.Parameters.Velocity	  := Mover_HMI.Parameters.Velocity;
	Mover.Parameters.Acceleration := Mover_HMI.Parameters.Acceleration;
	Mover.Parameters.Deceleration := Mover_HMI.Parameters.Deceleration;
	Mover.Parameters.Jerk		  := Mover_HMI.Parameters.Jerk;
	Mover.Parameters.Gap		  := Mover_HMI.Parameters.Gap;
	Mover.MoveToPosition(Position := Mover_HMI.Parameters.Position);
END_IF

Mover_HMI.Commands.MoveToStation.Permissive.Set(0, 'Mover not enabled', Mover.Enabled);
Mover_HMI.Commands.BumpCommand.Permissive.Set(0, 'Mover not enabled', Mover.Enabled);
BumpCommandRT(CLK := Mover_HMI.Commands.BumpCommand.Active);
IF BumpCommandRT.Q THEN
	Mover.Parameters.Velocity	  := Mover_HMI.Parameters.Velocity;
	Mover.Parameters.Acceleration := Mover_HMI.Parameters.Acceleration;
	Mover.Parameters.Deceleration := Mover_HMI.Parameters.Deceleration;
	Mover.Parameters.Jerk		  := Mover_HMI.Parameters.Jerk;
	Mover.Parameters.Gap		  := Mover_HMI.Parameters.Gap;
	Mover.MoveToPositionRelative(Distance := Mover_HMI.Parameters.Distance);
END_IF

Mover_HMI.Commands.Halt.Permissive.Set(0, 'Mover not enabled', Mover.Enabled);
HaltRt(Clk := Mover_Hmi.Commands.Halt.Active);
IF HaltRt.Q THEN
	Mover.Parameters.Jerk := Mover_Hmi.Parameters.Jerk;
	Mover.Halt(Deceleration := Mover_Hmi.Parameters.Deceleration, Gap := Mover_HMI.Parameters.Gap);
END_IF

ResetRT(Clk := Mover_HMI.Commands.Reset.Active);
IF ResetRT.Q THEN
	Mover.Reset();
END_IF
END_METHOD

(*FB_Init is always available implicitly and it is used primarily for initialization.
The return value is not evaluated. For a specific influence, you can also declare the
methods explicitly and provide additional code there with the standard initialization
code. You can evaluate the return value.*)
METHOD FB_Init : BOOL
VAR_INPUT
	(* TRUE: the retain variables are initialized (reset warm / reset cold)*)
	bInitRetains : BOOL;

	(* TRUE: the instance will be copied to the copy code afterward (online change)   *)
	bInCopyCode : BOOL;
	Name		: Core.T_MaxString;
	Mover		: I_XtsMover := 0; //If not set, the ControlObject MUST be set before being used
END_VAR
IF Mover <> 0 THEN
	THIS^.Mover	   := Mover;
	Mover_HMI.Name := Mover.Name;
END_IF

ControlType := 'XtsMover';
LinkObject	:= 'Mover_HMI';
END_METHOD

PROPERTY XtsMover : I_XtsMover
SET
Mover := XtsMover;
Mover_Hmi.Name := Mover.Name;
END_SET
END_PROPERTY

END_FUNCTION_BLOCK

// HMI/XtsStation_HMI
{attribute 'enable_dynamic_creation'}
FUNCTION_BLOCK XtsStation_HMI EXTENDS HmiFunction
VAR
	Station : I_XtsStation;
	{ attribute 'TcHmiSymbol.AddSymbol' }
	{ attribute 'TcHmiSymbol.AddSymbol.UserGroups' := '__SystemAdministrators,Admin' }
	Station_HMI : ST_XtsStation_HMI;
END_VAR

PROPERTY ControlObject : I_Base
SET
__QUERYINTERFACE(ControlObject, Station);
END_SET
END_PROPERTY

METHOD CyclicLogic
VAR_INST
	EnableRT	: R_TRIG;
	DisableRT	: R_TRIG;
	ClearLogRT	: R_TRIG;
	SetPosition : R_TRIG;
END_VAR
IF Station = 0 THEN
	RETURN;
END_IF

Station_HMI.Name				   := Station.Name;
Station_HMI.Enabled				   := Station.Enabled;
Station_HMI.MoverPresent		   := Station.MoverIsPresent;
Station_HMI.NumberMoversRegistered := Station.Status.NumberOfMoversRegistered;
Station_HMI.Position			   := Station.Position;
Station_HMI.LocalLog.Logs		   := Station.CommandLog.Commands;
ClearLogRT(Clk := Station_HMI.LocalLog.ClearLog);
IF ClearLogRT.Q THEN
	Station.CommandLog.Clear();
END_IF

IF NOT Station_Hmi.HmiEnabled THEN
	RETURN;
END_IF

SetPosition(Clk := Station_Hmi.SetPosition);
IF SetPosition.Q THEN
	Station.Position := Station_Hmi.TargetPosition;
END_IF

Station_Hmi.Enable.Permissive.Set(0, 'Station already enabled', NOT Station.Enabled);
EnableRT(Clk := Station_HMI.Enable.Active);
IF EnableRT.Q THEN
	Station.Enable();
END_IF

Station_Hmi.Disable.Permissive.Set(0, 'Station not enabled', Station.Enabled);
DisableRT(Clk := Station_HMI.Disable.Active);
IF DisableRT.Q THEN
	Station.Disable();
END_IF
END_METHOD

(*FB_Init is always available implicitly and it is used primarily for initialization.
The return value is not evaluated. For a specific influence, you can also declare the
methods explicitly and provide additional code there with the standard initialization
code. You can evaluate the return value.*)
METHOD FB_Init : BOOL
VAR_INPUT
	(* TRUE: the retain variables are initialized (reset warm / reset cold)*)
	bInitRetains : BOOL;

	(* TRUE: the instance will be copied to the copy code afterward (online change)   *)
	bInCopyCode : BOOL;
	Name		: Core.T_MaxString;
	Station		: I_XtsStation := 0; //If not set, the ControlObject MUST be set before being used
END_VAR
IF Station <> 0 THEN
	THIS^.Station	 := Station;
	Station_HMI.Name := Station.Name;
END_IF

ControlType := 'XtsStation';
LinkObject	:= 'Station_HMI';
END_METHOD

PROPERTY XtsStation : I_XtsStation
SET
Station := XtsStation;
Station_HMI.Name := Station.Name;
END_SET
END_PROPERTY

END_FUNCTION_BLOCK

// XtsStation/XtsStation
{attribute 'no_explicit_call' := 'This FB is a CLASS and must be accessed using methods or properties'}
FUNCTION_BLOCK XtsStation EXTENDS CyclicComponent IMPLEMENTS I_Base, I_XtsStation
VAR
	{attribute 'hide'}
	_Enabled : BOOL;
	{attribute 'hide'}
	_DefaultMoverlistBehavior : XtsMoverCollection;
	_RegisteredMovers		  : I_XtsMoverCollection := _DefaultMoverlistBehavior;
	{attribute 'hide'}
	_Status : XtsStationStatus(THIS^, _DefaultMoverMonitor);

	//
	_DefaultPositionBehavior : ReferencedPosition;
	_Position				 : I_Positionable := _DefaultPositionBehavior;

	//
	_DefaultMoverMonitor : MoverMonitorTask(THIS^, _RegisteredMovers);
	_MoverMonitor		 : I_MoverMonitor := _DefaultMoverMonitor;
	{attribute 'hide'}
	_LocalLogger : XtsLocalLogger;
	{attribute 'hide'}
	_Logger : XtsTracePublisher;
	{attribute 'hide'}
	LogMessage : TraceMessageInfo;
	{attribute 'hide'}
	LogSource : TraceSourceInfo;
END_VAR

//FB_Init is always available implicitly and it is used primarily for initialization.

//The return value is not evaluated. For a specific influence, you can also declare the

//methods explicitly and provide additional code there with the standard initialization

//code. You can evaluate the return value.
METHOD FB_Init : BOOL
VAR_INPUT
	bInitRetains : BOOL;				 // TRUE: the retain variables are initialized (reset warm / reset cold)
	bInCopyCode	 : BOOL;				 // TRUE: the instance will be copied to the copy code afterward (online change)
	Name		 : T_MaxString;			 //Name of the Station
	Position	 : LREAL;				 //Position in mm the Station will be located
	System		 : I_ContainXtsStations; //XtsSystem to self register to
END_VAR
_Position.Position	 := Position;
LogSource.SourceName := Name;
IF System <> 0 THEN
	System.Stations.AddItem(THIS^);
	RegisterWithParent(System);
END_IF

_Status.SetRegisteredMovers(_RegisteredMovers);
_Logger.Subscribe(_LocalLogger);
IF XtsCoreParameters.TcEventLoggerEnabled THEN
	_Logger.Subscribe(XtsTrace.EventLogger);
END_IF
END_METHOD

//Disable the station
METHOD Disable
VAR
	LogMessage : TraceMessageInfo;
	LogSource  : TraceSourceInfo;
END_VAR
_Enabled := FALSE;
LogSource.SourceName := _Name;
LogMessage.Message	 := 'Disabled.';
LogMessage.MessageId := E_XtsLogMessage.StationDisabled;
_Logger.LogMessageInstance(LogSource, LogMessage);
END_METHOD

//Enable the station
METHOD Enable
VAR
	LogMessage : TraceMessageInfo;
	LogSource  : TraceSourceInfo;
END_VAR
_Enabled			 := TRUE;
LogSource.SourceName := _Name;
LogMessage.Message	 := 'Enabled.';
LogMessage.MessageId := E_XtsLogMessage.StationEnabled;
_Logger.LogMessageInstance(LogSource, LogMessage);
END_METHOD

{attribute 'monitoring' := 'call'}
PROPERTY Enabled : BOOL
GET
Enabled := _Enabled;
END_GET
END_PROPERTY

{attribute 'monitoring':='call'}
PROPERTY CommandLog : I_XtsLocalLog
GET
CommandLog := _LocalLogger;
END_GET
END_PROPERTY

PROPERTY TracePublisher : I_XtsTracePublisher
GET
TracePublisher := _Logger;
END_GET
END_PROPERTY

METHOD AcceptStationVisitor
VAR_INPUT
	StationVisitor : I_XtsStationVisitor;
END_VAR
StationVisitor.VisitStation(THIS^);
END_METHOD

METHOD CyclicLogic
IF NOT _Enabled THEN
	RETURN;
END_IF
_MoverMonitor.CyclicLogic();
END_METHOD

//Deregisters Mover to be Monitored by Station
METHOD DeregisterMover
VAR_INPUT
	Mover : I_XtsMover; //Mover to Deregister
END_VAR
_RegisteredMovers.Remove(Mover);
LogSource.SourceName := _Name;
LogMessage.Message	 := CONCAT('Mover Deregistered: ', Mover.Name);
LogMessage.Severity	 := 0;
LogMessage.MessageId := E_XtsLogMessage.StationMoverDeregistered;
_Logger.LogMessageInstance(LogSource, LogMessage);
END_METHOD

//Gets the Current Mover latched at the Station
METHOD GetMover : I_XtsMover
VAR_INPUT
END_VAR

VAR
	_Mover	   : I_XtsMover;
	LogMessage : TraceMessageInfo;
	LogSource  : TraceSourceInfo;
END_VAR
_Mover				 := _MoverMonitor.GetMover();
LogSource.SourceName := _Name;
LogMessage.Message	 := CONCAT('Get Mover called: ', _Mover.Name);
LogMessage.Severity	 := 10;
LogMessage.MessageId := E_XtsLogMessage.StationGetMoverCalled;
_Logger.LogMessageInstance(LogSource, LogMessage);
GetMover := _Mover;
END_METHOD

//Checks if provided Mover is registered and monitored
METHOD IsMoverRegistered : BOOL
VAR_INPUT
	Mover : I_XtsMover; //Mover to check
END_VAR
_RegisteredMovers.ResetIterator();
WHILE _RegisteredMovers.MoveToNext DO
	IF _RegisteredMovers.Current = Mover THEN
		IsMoverRegistered := TRUE;
		RETURN;
	END_IF
END_WHILE
END_METHOD

{attribute 'monitoring' := 'call'}
//Signal for if a Mover has arrived at the Station.
PROPERTY MoverIsPresent : BOOL
GET
MoverIsPresent := _MoverMonitor.MoverPresent;
END_GET
END_PROPERTY

//Currently registered and monitored Movers
PROPERTY Movers : I_XtsMoverEnumerator
GET
Movers := _RegisteredMovers;
END_GET
END_PROPERTY

{attribute 'monitoring' := 'call'}
//Location of the Station in mm
PROPERTY Position : LREAL
GET
Position := _Position.Position;
END_GET
SET
_Position.Position := Position;
END_SET
END_PROPERTY

//Registers Mover to be Monitored by Station
METHOD RegisterMover
VAR_INPUT
	Mover : I_XtsMover; //Mover to regsiter
END_VAR

VAR
	found	   : BOOL;
END_VAR
_RegisteredMovers.ResetIterator();
WHILE _RegisteredMovers.MoveToNext DO
	found := _RegisteredMovers.Current = Mover;
	IF found THEN
		RETURN;
	END_IF
END_WHILE

_RegisteredMovers.AddItem(Mover);
LogSource.SourceName := _Name;
LogMessage.Message	 := CONCAT('Mover Registered: ', Mover.Name);
LogMessage.Severity	 := 0;
LogMessage.MessageId := E_XtsLogMessage.StationMoverRegistered;
_Logger.LogMessageInstance(LogSource, LogMessage);
END_METHOD

{attribute 'monitoring':='call'}
PROPERTY Status : I_XtsStationStatus
GET
Status := _Status;
END_GET
END_PROPERTY

END_FUNCTION_BLOCK

// HMI/XtsPositionTrigger_HMI
FUNCTION_BLOCK XtsPositionTrigger_HMI EXTENDS HmiFunction
VAR
	PositionTrigger : I_XtsPositionTrigger;
	{ attribute 'TcHmiSymbol.AddSymbol' }
	{ attribute 'TcHmiSymbol.AddSymbol.UserGroups' := '__SystemAdministrators,Admin' }
	PositionTrigger_HMI : ST_XtsPositionTrigger_HMI;
END_VAR

PROPERTY ControlObject : I_Base
SET
__QUERYINTERFACE(ControlObject, PositionTrigger);
END_SET
END_PROPERTY

METHOD CyclicLogic
VAR_INST
	EnableRT	 : R_TRIG;
	DisableRT	 : R_TRIG;
	ClearLogRT	 : R_TRIG;
	ClearQueueRT : R_TRIG;
	SetPosition : R_TRIG;
END_VAR
IF PositionTrigger = 0 THEN
	RETURN;
END_IF

PositionTrigger_HMI.Name				   := PositionTrigger.Name;
PositionTrigger_HMI.Enabled				   := PositionTrigger.Enabled;
PositionTrigger_HMI.MoverPresent		   := PositionTrigger.MoverIsPresent;
PositionTrigger_HMI.NumberMoversRegistered := PositionTrigger.Status.NumberOfMoversRegistered;
PositionTrigger_HMI.Position			   := PositionTrigger.Position;
PositionTrigger_HMI.LocalLog.Logs		   := PositionTrigger.CommandLog.Commands;
PositionTrigger_HMI.NumberEventsInQueue	   := PositionTrigger.MoverQueue.Count;
ClearLogRT(Clk := PositionTrigger_HMI.LocalLog.ClearLog);
IF ClearLogRT.Q THEN
	PositionTrigger.CommandLog.Clear();
END_IF

IF NOT PositionTrigger_Hmi.HmiEnabled THEN
	RETURN;
END_IF

SetPosition(Clk := PositionTrigger_HMI.SetPosition);
IF SetPosition.Q THEN
	PositionTrigger.Position := PositionTrigger_HMI.TargetPosition;
END_IF

PositionTrigger_HMI.Enable.Permissive.Set(0, 'Trigger already enabled', NOT PositionTrigger.Enabled);
EnableRT(Clk := PositionTrigger_HMI.Enable.Active);
IF EnableRT.Q THEN
	PositionTrigger.Enable();
END_IF

PositionTrigger_HMI.Disable.Permissive.Set(0, 'Trigger not enabled', PositionTrigger.Enabled);
DisableRT(Clk := PositionTrigger_HMI.Disable.Active);
IF DisableRT.Q THEN
	PositionTrigger.Disable();
END_IF

ClearQueueRT(Clk := PositionTrigger_HMI.ClearQueue.Active);
IF ClearQueueRT.Q THEN
	PositionTrigger.MoverQueue.Clear();
END_IF
END_METHOD

(*FB_Init is always available implicitly and it is used primarily for initialization.
The return value is not evaluated. For a specific influence, you can also declare the
methods explicitly and provide additional code there with the standard initialization
code. You can evaluate the return value.*)
METHOD FB_Init : BOOL
VAR_INPUT
	(* TRUE: the retain variables are initialized (reset warm / reset cold)*)
	bInitRetains : BOOL;

	(* TRUE: the instance will be copied to the copy code afterward (online change)   *)
	bInCopyCode		: BOOL;
	Name			: Core.T_MaxString;
	PositionTrigger : I_XtsPositionTrigger := 0; //If not set, the ControlObject MUST be set before being used
END_VAR
IF PositionTrigger <> 0 THEN
	THIS^.PositionTrigger	 := PositionTrigger;
	PositionTrigger_HMI.Name := PositionTrigger.Name;
END_IF

ControlType := 'XtsPositionTrigger';
LinkObject	:= 'PositionTrigger_HMI';
END_METHOD

PROPERTY XtsPositionTrigger : I_XtsPositionTrigger
SET
PositionTrigger := XtsPositionTrigger;
PositionTrigger_HMI.Name := PositionTrigger.Name;
END_SET
END_PROPERTY

END_FUNCTION_BLOCK

// HMI/XtsZone_HMI
FUNCTION_BLOCK XtsZone_HMI EXTENDS HmiFunction
VAR
	Zone : I_XtsZone;
	{ attribute 'TcHmiSymbol.AddSymbol' }
	{ attribute 'TcHmiSymbol.AddSymbol.UserGroups' := '__SystemAdministrators,Admin' }
	Zone_HMI : ST_XtsZone_HMI;
END_VAR

PROPERTY ControlObject : I_Base
SET
__QUERYINTERFACE(ControlObject, Zone);
END_SET
END_PROPERTY

METHOD CyclicLogic
VAR_INST
	SortedMoverRT	 : R_TRIG;
	ClearLogRT		 : R_TRIG;
	EnableRT		 : R_TRIG;
	DisableRT		 : R_TRIG;
	MoveToPositionRT : R_TRIG;
	MoveVelocityRT	 : R_TRIG;
	MoveToStationRT	 : R_TRIG;
	HaltRt			 : R_TRIG;

	//
	Commands : XtsMoverCommander;
END_VAR
IF Zone = 0 THEN
	RETURN;
END_IF

Zone_HMI.Name					 := Zone.Name;
Zone_HMI.StartPosition			 := Zone.StartPosition;
Zone_HMI.EndPosition			 := Zone.EndPosition;
Zone_HMI.NumberMoversInZone		 := Zone.Status.NumberOfMoversInZone;
Zone_HMI.LocalLog.Logs			 := Zone.CommandLog.Commands;
Commands.Parameters.Position	 := Zone_Hmi.CommandParameters.Velocity;
Commands.Parameters.Velocity	 := Zone_Hmi.CommandParameters.Velocity;
Commands.Parameters.Acceleration := Zone_Hmi.CommandParameters.Acceleration;
Commands.Parameters.Deceleration := Zone_Hmi.CommandParameters.Deceleration;
Commands.Parameters.Jerk		 := Zone_Hmi.CommandParameters.Jerk;
Commands.Parameters.Gap			 := Zone_Hmi.CommandParameters.Gap;
ClearLogRT(Clk := Zone_HMI.LocalLog.ClearLog);
IF ClearLogRT.Q THEN
	Zone.CommandLog.Clear();
END_IF

IF NOT Zone_HMI.HmiEnabled THEN
	RETURN;
END_IF

Zone_HMI.GetSortedMover.Permissive.Set(0, 'No Movers in Zone', Zone.Status.NumberOfMoversInZone = 0);
Zone_HMI.GetSortedMover.Permissive.Set(1, 'Index outside range Zone', Zone_Hmi.SortedPosition < 0 OR Zone_Hmi.SortedPosition >= Zone.Status.NumberOfMoversInZone);
SortedMoverRT(Clk := Zone_HMI.GetSortedMover.Active);
IF SortedMoverRT.Q THEN
	Zone_HMI.SortedMover := Zone.GetSortedMover(Zone_Hmi.SortedPosition, Zone_Hmi.SortedDirection).Name;
END_IF

EnableRT(Clk := Zone_Hmi.MoverCommands.Enable.Active);
IF EnableRT.Q THEN
	Commands.Enable(Zone);
END_IF

DisableRT(Clk := Zone_Hmi.MoverCommands.Disable.Active);
IF DisableRT.Q THEN
	Commands.Disable(Zone);
END_IF

MoveVelocityRT(Clk := Zone_Hmi.MoverCommands.MoveVelocity.Active);
IF MoveVelocityRT.Q THEN
	Commands.MoveVelocity(Visitee := Zone, Velocity := Zone_Hmi.CommandParameters.Velocity, Direction := Commands.Parameters.Direction);
END_IF

MoveToPositionRT(Clk := Zone_Hmi.MoverCommands.MoveToPosition.Active);
IF MoveToPositionRT.Q THEN
	Commands.MoveToPosition(Visitee := Zone, Position := Zone_Hmi.CommandParameters.Position, Direction := Commands.Parameters.Direction);
END_IF

HaltRt(Clk := Zone_Hmi.MoverCommands.Halt.Active);
IF HaltRt.Q THEN
	Commands.Halt(Visitee := Zone, Deceleration := Zone_Hmi.CommandParameters.Deceleration, Gap := Zone_Hmi.CommandParameters.Gap);
END_IF
END_METHOD

(*FB_Init is always available implicitly and it is used primarily for initialization.
The return value is not evaluated. For a specific influence, you can also declare the
methods explicitly and provide additional code there with the standard initialization
code. You can evaluate the return value.*)
METHOD FB_Init : BOOL
VAR_INPUT
	(* TRUE: the retain variables are initialized (reset warm / reset cold)*)
	bInitRetains : BOOL;

	(* TRUE: the instance will be copied to the copy code afterward (online change)   *)
	bInCopyCode : BOOL;
	Name		: Core.T_MaxString;
	Zone		: I_XtsZone := 0; //If not set, the ControlObject MUST be set before being used
END_VAR
IF Zone <> 0 THEN
	THIS^.Zone	  := Zone;
	Zone_HMI.Name := Zone.Name;
END_IF

ControlType := 'XtsZone';
LinkObject	:= 'Zone_HMI';
END_METHOD

END_FUNCTION_BLOCK

// HMI/XtsSystem_HMI
FUNCTION_BLOCK XtsSystem_HMI EXTENDS HmiFunction
VAR
	System : I_XtsSystem;
	{ attribute 'TcHmiSymbol.AddSymbol' }
	{ attribute 'TcHmiSymbol.AddSymbol.UserGroups' := '__SystemAdministrators,Admin' }
	System_HMI : ST_XtsSystem_HMI;
END_VAR

PROPERTY ControlObject : I_Base
SET
__QUERYINTERFACE(ControlObject, System);
END_SET
END_PROPERTY

METHOD CyclicLogic
VAR_INST
	EnableRT   : R_TRIG;
	DisableRT  : R_TRIG;
	ResetRT	   : R_Trig;
	ClearLogRT : R_TRIG;
END_VAR
IF System = 0 THEN
	RETURN;
END_IF

IF System_HMI.CurrentTask <> System.CurrentTask.TaskName THEN
	System_HMI.LastTask	   := System_HMI.CurrentTask;
	System_HMI.CurrentTask := System.CurrentTask.TaskName;
END_IF

System_HMI.Name						:= System.Name;
System_HMI.Enabled					:= System.Enabled;
System_HMI.ErrorId					:= TO_STRING(System.ErrorId);
System_HMI.HasError					:= System.Error;
System_HMI.Initialized				:= System.Initialized;
System_HMI.MoversEnabled			:= System.MoversEnabled;
System_HMI.CaGroup					:= TO_STRING(System.CaGroupStatus);
System_HMI.MoverType				:= System.UtilityProperties.Mover.XtsMoverType;
System_HMI.NumberOfStations			:= System.Status.NumberOfStations;
System_HMI.NumberOfPositionTriggers := System.Status.NumberOfPositionTriggers;
System_HMI.NumberOfMovers			:= System.Status.NumberOfMovers;
System_HMI.NumberOfParts			:= System.Status.NumberOfParts;
System_HMI.NumberOfTracks			:= System.Status.NumberOfTracks;
System_HMI.NumberOfZones			:= System.Status.NumberOfZones;
System_HMI.Simulated				:= System.Status.Simulated;
System_HMI.Vdc24Okay				:= System.Status.Vdc24Okay;
System_HMI.Vdc48Okay				:= System.Status.Vdc48Okay;
System_HMI.LocalLog.Logs			:= System.CommandLog.Commands;
//Commands from HMI are locked if the HMI is not enabled
IF NOT System_HMI.HmiEnabled THEN
	RETURN;
END_IF

ClearLogRT(Clk := System_HMI.LocalLog.ClearLog);
IF ClearLogRT.Q THEN
	System.CommandLog.Clear();
END_IF

EnableRT(Clk := System_HMI.Enable);
IF EnableRT.Q THEN
	System.Enable();
END_IF

DisableRT(Clk := System_HMI.Disable);
IF DisableRT.Q THEN
	System.Disable();
END_IF

ResetRT(Clk := System_HMI.Reset);
IF ResetRT.Q THEN
	System.Reset();
END_IF
END_METHOD

(*FB_Init is always available implicitly and it is used primarily for initialization.
The return value is not evaluated. For a specific influence, you can also declare the
methods explicitly and provide additional code there with the standard initialization
code. You can evaluate the return value.*)
METHOD FB_Init : BOOL
VAR_INPUT
	(* TRUE: the retain variables are initialized (reset warm / reset cold)*)
	bInitRetains : BOOL;

	(* TRUE: the instance will be copied to the copy code afterward (online change)   *)
	bInCopyCode : BOOL;
	Name		: Core.T_MaxString;
	System		: I_XtsSystem := 0; //If not set, the ControlObject MUST be set before being used
END_VAR
IF System <> 0 THEN
	THIS^.System	:= System;
	System_HMI.Name := System.Name;
END_IF

ControlType := 'XtsSystem';
LinkObject	:= 'System_HMI';
END_METHOD

END_FUNCTION_BLOCK

// HMI/XtsModule_HMI
FUNCTION_BLOCK XtsModule_HMI EXTENDS HmiFunction
VAR
	_Module : I_XtsModule;
	{ attribute 'TcHmiSymbol.AddSymbol' }
	{ attribute 'TcHmiSymbol.AddSymbol.UserGroups' := '__SystemAdministrators,Admin' }
	Module_HMI : ST_XtsModule_HMI;
END_VAR

PROPERTY ControlObject : I_Base
SET
__QUERYINTERFACE(ControlObject, _Module);
END_SET
END_PROPERTY

METHOD CyclicLogic
IF _Module = 0 THEN
	RETURN;
END_IF

Module_HMI.ModuleReady := _Module.ModuleReady;
END_METHOD

(*FB_Init is always available implicitly and it is used primarily for initialization.
The return value is not evaluated. For a specific influence, you can also declare the
methods explicitly and provide additional code there with the standard initialization
code. You can evaluate the return value.*)
METHOD FB_Init : BOOL
VAR_INPUT
	(* TRUE: the retain variables are initialized (reset warm / reset cold)*)
	bInitRetains : BOOL;

	(* TRUE: the instance will be copied to the copy code afterward (online change)   *)
	bInCopyCode : BOOL;
	Name		: Core.T_MaxString;
	XtsModule	: I_XtsModule := 0; //If not set, the ControlObject MUST be set before being used
END_VAR
IF XtsModule <> 0 THEN
	THIS^._Module	:= XtsModule;
	Module_HMI.Name := XtsModule.Name;
END_IF
ControlType := 'XtsModule';
LinkObject	:= 'Module_HMI';
END_METHOD

PROPERTY XtsModule : I_XtsModule
SET
_Module			:= XtsModule;
Module_Hmi.Name := _Module.Name;
END_SET
END_PROPERTY

END_FUNCTION_BLOCK

// HMI/XtsPart_HMI
FUNCTION_BLOCK XtsPart_HMI EXTENDS HmiFunction
VAR
	Part : I_XtsPart;
	{ attribute 'TcHmiSymbol.AddSymbol' }
	{ attribute 'TcHmiSymbol.AddSymbol.UserGroups' := '__SystemAdministrators,Admin' }
	Part_HMI : ST_XtsPart_HMI;
END_VAR

PROPERTY ControlObject : I_Base
SET
__QUERYINTERFACE(ControlObject, Part);
END_SET
END_PROPERTY

METHOD CyclicLogic
IF Part = 0 THEN
	RETURN;
END_IF

Part_HMI.PartReady := Part.PartReady;
Part_HMI.Id		   := Part.XtsPartId;
END_METHOD

(*FB_Init is always available implicitly and it is used primarily for initialization.
The return value is not evaluated. For a specific influence, you can also declare the
methods explicitly and provide additional code there with the standard initialization
code. You can evaluate the return value.*)
METHOD FB_Init : BOOL
VAR_INPUT
	(* TRUE: the retain variables are initialized (reset warm / reset cold)*)
	bInitRetains : BOOL;

	(* TRUE: the instance will be copied to the copy code afterward (online change)   *)
	bInCopyCode : BOOL;
	Name		: Core.T_MaxString;
	Part		: I_XtsPart := 0; //If not set, the ControlObject MUST be set before being used
END_VAR
IF Part <> 0 THEN
	THIS^.Part	  := Part;
	Part_HMI.Name := Part.Name;
END_IF

ControlType := 'XtsPart';
LinkObject	:= 'Part_HMI';
END_METHOD

PROPERTY XtsPart : I_XtsPart
SET
Part := XtsPart;
Part_HMI.Name := Part.Name;
END_SET
END_PROPERTY

END_FUNCTION_BLOCK

// Project Information/F_GetCompany
// This function has been automatically generated from the project information.
{attribute 'signature_flag' := '1073741824'}
{attribute 'TcGenerated'}
{attribute 'no-analysis'}
FUNCTION F_GetCompany : WSTRING
VAR_INPUT
	
END_VAR

F_GetCompany := "Beckhoff Automation LLC";

END_FUNCTION

// Project Information/F_GetTitle
// This function has been automatically generated from the project information.
{attribute 'signature_flag' := '1073741824'}
{attribute 'TcGenerated'}
{attribute 'no-analysis'}
FUNCTION F_GetTitle : WSTRING
VAR_INPUT
	
END_VAR

F_GetTitle := "XtsCore";

END_FUNCTION

// Project Information/F_GetVersion
// This function has been automatically generated from the project information.
{attribute 'signature_flag' := '1073741824'}
{attribute 'TcGenerated'}
{attribute 'no-analysis'}
FUNCTION F_GetVersion : ST_LibVersion
VAR_INPUT
	
END_VAR

F_GetVersion.iMajor := 0;
F_GetVersion.iMinor := 12;
F_GetVersion.iBuild := 1;
F_GetVersion.iRevision := 23;
F_GetVersion.sVersion := '0.12.1.23';
F_GetVersion.nFlags := 0;

END_FUNCTION

// Utilities/Validators/AllMoversValidator
FUNCTION_BLOCK AllMoversValidator IMPLEMENTS I_XtsMoverValidator
VAR
END_VAR

METHOD Valid : BOOL
VAR_INPUT
	Mover	: I_XtsMover;
END_VAR
Valid := TRUE;
END_METHOD

END_FUNCTION_BLOCK

// Utilities/Validators/NoMoversValidator
FUNCTION_BLOCK NoMoversValidator IMPLEMENTS I_XtsMoverValidator
VAR
END_VAR

METHOD Valid : BOOL
VAR_INPUT
	Mover	: I_XtsMover;
END_VAR
Valid := FALSE;
END_METHOD

END_FUNCTION_BLOCK

// Utilities/IsNullObject
FUNCTION IsNullObject : BOOL
VAR_INPUT
	Object : I_Base;
END_VAR
VAR
	NullObject : I_NullObject;
END_VAR

IsNullObject := __QUERYINTERFACE(Object,NullObject);

END_FUNCTION

// Utilities/IsValidObject
FUNCTION IsValidObject : BOOL
VAR_INPUT
	Object : I_Base;
END_VAR
VAR
	value : BOOL;
	inverse : BOOL;
	NullObject : I_NullObject;
END_VAR

IsValidObject := (NOT __QUERYINTERFACE(Object, NullObject));

END_FUNCTION

// XtsStation/Interfaces/I_MoverPositionMonitor
INTERFACE I_MoverPositionMonitor EXTENDS I_Base

END_INTERFACE
